{attribute addProperty BoxType "EPP2308-0001-0016"}
{attribute addProperty Id "ChannelAT %I*ARRAY[0..3] OF Channel_E4AEF59E3240Channel_1AT %Q*ARRAY[0..3] OF Channel_7F374EB03240WcStateAT %I*WcState_F855686C1620InfoDataAT %I*InfoData_192954DE1620"}
{attribute addProperty CRC "2032139953"}
{attribute addProperty SizeInBites "96"}
{attribute addProperty SizeInBytes "12"}
TYPE EPP2308_E5848397 :
STRUCT
	{attribute addProperty Name "Channel"}
	Channel : ARRAY[0..3] OF Channel_E4AEF59E;
	{attribute addProperty Name "Channel_1"}
	Channel_1 : ARRAY[0..3] OF Channel_7F374EB0;
	{attribute addProperty Name "WcState"}
	WcState : WcState_F855686C;
	{attribute addProperty Name "InfoData"}
	InfoData : InfoData_192954DE;
END_STRUCT
END_TYPE

(* stored: Version 1.2.0.0, ProductVersion 3.1.4024.9
   DUT EPP2308_E5848397: Id {0ed35d55-3fff-4669-87b7-94dfe6cbd533} *)
